// TwinCAT 3 PLC project Untitled1
// ProgramVersion: 3.1.4023.0
// libraries:
//   Tc2_Standard, * (Beckhoff Automation GmbH)
//   Tc2_System, * (Beckhoff Automation GmbH)
//   Tc3_Module, * (Beckhoff Automation GmbH)
// project tree:
//   DUTs/ ST_Banner_K30PTKQ_Control.TcDUT, ST_Banner_K30PTKQ_Status.TcDUT, ST_Keyence_LRXH100_Status.TcDUT, ST_Balluff_BMF00LA_Status.TcDUT
//   FBs/ FB_Banner_K30PTKQ.TcPOU, FB_Keyence_LRXH100.TcPOU, FB_Balluff_BMF00LA.TcPOU
//   / PlcTask.TcTTO
//   POUs/ MAIN.TcPOU

CONFIGURATION Untitled1
    RESOURCE PLC ON TwinCAT3
        TASK PlcTask(INTERVAL := T#10ms, PRIORITY := 20);
        PROGRAM MAIN WITH PlcTask : MAIN;
    END_RESOURCE
END_CONFIGURATION

// ---- DUTs/ST_Banner_K30PTKQ_Control.TcDUT
(*
	This structure contains all the inputs of the BANNER LED.
	The inputs and the outputs are linked to the device as well.
*)

TYPE ST_Banner_K30PTKQ_Control :
	STRUCT
	Color1					: UINT; (* 0 = Green, 1 = Red, 2 = Orange, 3 = Amber, 4 = Yellow,
									5 = Lime Green, 6 = Spring Green, 7 = Cyan, 8 = Sky Blue,
									9 = Blue, 10 = Violet, 11 = Magenta, 12 = Rose, 13 = White,
									14 = Custom1, 15 = Custom2 *)
	Color2					: UINT; (* 0 = Green, 1 = Red, 2 = Orange, 3 = Amber, 4 = Yellow,
									5 = Lime Green, 6 = Spring Green, 7 = Cyan, 8 = Sky Blue,
									9 = Blue, 10 = Violet, 11 = Magenta, 12 = Rose, 13 = White,
									14 = Custom1, 15 = Custom2 *)
	Color1Intensity			: UINT; (* 0 = High, 1 = Medium, 2 = Low, 3 = Off, 4 = Custom *)
	Color2Intensity			: UINT; (* 0 = High, 1 = Medium, 2 = Low, 3 = Off, 4 = Custom *)
	SequenceStartLocation	: UINT; (* 0 = LED1, 1 = LED2, 2 = LED3, 3 = LED4 *)
	DynamicSequenceValue	: UINT; (* 0-255 *)
	AnimationSpeed			: UINT; (* 0 = Slow, 1 = Medium, 2 = Fast, 3 = Custom *)
	Reserved				: UINT; (* Reserved *)
	AnimationType			: UINT; (* 0 = Off, 1 = Steady, 2 = Flash, 3 = Two Color Flash,
									   4 = 50/50, 5 = 50/50 Rotate, 6 = Chase, 7 = Intensity Sweep,
									   8 = Color Sweep, 9 = Sequence, 10 = Wave, 11 = Double Wave *)
	AnimationDirection		: UINT; (* 0 = CCW, 1 = CW *)
	AnimationPattern		: UINT; (* 0 = Flash, 1 = Strobe, 2 = Three Pulse, 3 = SOS, 4 = Random *)
	END_STRUCT
END_TYPE

// ---- DUTs/ST_Banner_K30PTKQ_Status.TcDUT
(*
	This structure contains all the outputs of the BANNER LED.
	The inputs and the outputs are linked to the device as well.
*)
TYPE ST_Banner_K30PTKQ_Status :
	STRUCT
	OutputState	: UINT; (* 0 = Normally Closed, 1 = Normally Open *)
	END_STRUCT
END_TYPE

// ---- DUTs/ST_Keyence_LRXH100_Status.TcDUT
(*
	This structure contains all the outputs of the BANNER LED.
	The inputs and the outputs are linked to the device as well.
*)
TYPE ST_Keyence_LRXH100_Status :
STRUCT
	CurrentValue		: INT; (* The distance from the target -9999 to 10001 *)
	ErrorOvercurrent	: BOOL; (* 0x7710 An overcurrent error has occurred. *)
	ErrorHeadError		: BOOL; (* 0x1803 A laser fault has occurred. *)
	ErrorEepromError	: BOOL; (* 0x5000 An EEPROM error has occurred in the sensor. *)
	Error17Error		: BOOL; (* 0x1807 Error 1 - 7 *)
	Output1				: BOOL; (* Output 1 *)
	Output2				: BOOL; (* Output 2 *)
	Warning				: BOOL; (* Warning *)
END_STRUCT
END_TYPE

// ---- DUTs/ST_Balluff_BMF00LA_Status.TcDUT
(*
	This structure contains all the outputs of the BANNER LED.
	The inputs and the outputs are linked to the device as well.
*)
TYPE ST_Balluff_BMF00LA_Status :
STRUCT
	Stability	: BOOL; (* Monitor if the sensor recognises a signal *)
	TeachIn		: BOOL; (* Monitor whether it is currently being taught *)
	BDC1		: BOOL; (* Setted point 1 *)
	BDC2		: BOOL; (* Setted point 2 *)
	BDC3		: BOOL; (* Setted point 3 *)
	BDC4		: BOOL; (* Setted point 4 *)
	BDC5		: BOOL; (* Setted point 5 *)
	BDC6		: BOOL; (* Setted point 6 *)
	BDC7		: BOOL; (* Setted point 7 *)
	BDC8		: BOOL; (* Setted point 8 *)
END_STRUCT
END_TYPE

// ---- POUs/MAIN.TcPOU
PROGRAM MAIN
VAR
{attribute 'TcLinkToOSO' := '.In.OutputState 			:= <0,1,0>TIID^Device 2 (EtherCAT)^Box 1 (EP6228-0022)^Banner_K30PTKQ^In^Output State;
							 .Out.Color1 	 			:= <0,5,0>TIID^Device 2 (EtherCAT)^Box 1 (EP6228-0022)^Banner_K30PTKQ^Out^Color 1;
							 .Out.Color2 	 			:= <0,5,0>TIID^Device 2 (EtherCAT)^Box 1 (EP6228-0022)^Banner_K30PTKQ^Out^Color 2;
							 .Out.Color1Intensity 	 	:= <0,3,0>TIID^Device 2 (EtherCAT)^Box 1 (EP6228-0022)^Banner_K30PTKQ^Out^Color 1 Intensity;
							 .Out.Color2Intensity 	 	:= <0,3,0>TIID^Device 2 (EtherCAT)^Box 1 (EP6228-0022)^Banner_K30PTKQ^Out^Color 2 Intensity;
							 .Out.SequenceStartLocation	:= <0,3,0>TIID^Device 2 (EtherCAT)^Box 1 (EP6228-0022)^Banner_K30PTKQ^Out^Sequence Start Location;
							 .Out.DynamicSequenceValue 	:= <0,8,0>TIID^Device 2 (EtherCAT)^Box 1 (EP6228-0022)^Banner_K30PTKQ^Out^Dynamic Sequence Value (0-255);
							 .Out.AnimationSpeed 	 	:= <0,2,0>TIID^Device 2 (EtherCAT)^Box 1 (EP6228-0022)^Banner_K30PTKQ^Out^Animation Speed;
							 .Out.Reserved 	 			:= <0,2,0>TIID^Device 2 (EtherCAT)^Box 1 (EP6228-0022)^Banner_K30PTKQ^Out^Reserved;
							 .Out.AnimationType 	 	:= <0,4,0>TIID^Device 2 (EtherCAT)^Box 1 (EP6228-0022)^Banner_K30PTKQ^Out^Animation Type;
							 .Out.AnimationDirection 	:= <0,1,0>TIID^Device 2 (EtherCAT)^Box 1 (EP6228-0022)^Banner_K30PTKQ^Out^Animation Direction;
							 .Out.AnimationPattern 	 	:= <0,3,0>TIID^Device 2 (EtherCAT)^Box 1 (EP6228-0022)^Banner_K30PTKQ^Out^Animation Pattern'}	
	LED		: FB_Banner_K30PTKQ; (*This is an instance of the FB_LED Funciton block*)
	{attribute 'TcLinkTo' := '.In.Stability 			:= TIID^Device 2 (EtherCAT)^Box 1 (EP6228-0022)^Balluff_BMF00LA^In^Stability;
							  .In.TeachIn 				:= TIID^Device 2 (EtherCAT)^Box 1 (EP6228-0022)^Balluff_BMF00LA^In^Teach-In;
							  .In.BDC1 					:= TIID^Device 2 (EtherCAT)^Box 1 (EP6228-0022)^Balluff_BMF00LA^In^BDC1;
							  .In.BDC2 					:= TIID^Device 2 (EtherCAT)^Box 1 (EP6228-0022)^Balluff_BMF00LA^In^BDC2;
							  .In.BDC3 					:= TIID^Device 2 (EtherCAT)^Box 1 (EP6228-0022)^Balluff_BMF00LA^In^BDC3;
							  .In.BDC4 					:= TIID^Device 2 (EtherCAT)^Box 1 (EP6228-0022)^Balluff_BMF00LA^In^BDC4;
							  .In.BDC5 					:= TIID^Device 2 (EtherCAT)^Box 1 (EP6228-0022)^Balluff_BMF00LA^In^BDC5;
							  .In.BDC6 					:= TIID^Device 2 (EtherCAT)^Box 1 (EP6228-0022)^Balluff_BMF00LA^In^BDC6;
							  .In.BDC7 					:= TIID^Device 2 (EtherCAT)^Box 1 (EP6228-0022)^Balluff_BMF00LA^In^BDC7;
							  .In.BDC8 					:= TIID^Device 2 (EtherCAT)^Box 1 (EP6228-0022)^Balluff_BMF00LA^In^BDC8'}
	Sensor	: FB_Balluff_BMF00LA; (*This is an instance of the FB_Sensor Funciton block*)
	
	{attribute 'TcLinkTo' := '.In.CurrentValue 			:= TIID^Device 2 (EtherCAT)^Box 1 (EP6228-0022)^Keyence_LRXH100^In^Current Value;
							  .In.ErrorOvercurrent 		:= TIID^Device 2 (EtherCAT)^Box 1 (EP6228-0022)^Keyence_LRXH100^In^Error : Overcurrent;
						      .In.ErrorHeadError	 	:= TIID^Device 2 (EtherCAT)^Box 1 (EP6228-0022)^Keyence_LRXH100^In^Error : Head Error;
							  .In.ErrorEepromError 	 	:= TIID^Device 2 (EtherCAT)^Box 1 (EP6228-0022)^Keyence_LRXH100^In^Error : EEPROM Error;
							  .In.Error17Error 			:= TIID^Device 2 (EtherCAT)^Box 1 (EP6228-0022)^Keyence_LRXH100^In^Error : Error 1 - 7;
							  .In.Output1 	 			:= TIID^Device 2 (EtherCAT)^Box 1 (EP6228-0022)^Keyence_LRXH100^In^Output 1;
							  .In.Output2	 	 		:= TIID^Device 2 (EtherCAT)^Box 1 (EP6228-0022)^Keyence_LRXH100^In^Output 2;
							  .In.Warning 	 			:= TIID^Device 2 (EtherCAT)^Box 1 (EP6228-0022)^Keyence_LRXH100^In^Warning'}
	KeyenceSensor			: FB_Keyence_LRXH100; (*This is an instance of the FB_Keyence Funciton block*)
END_VAR
VAR
	sVendorName				: STRING(64);
	sVendorText				: STRING(64);
	bTrig					: BOOL;
	fbAdsRead				: Tc2_System.ADSREAD;
	i						: INT;
	sData					: ARRAY[0..3] OF STRING(64);
	nIndexOffset			: ARRAY[0..3] OF UDINT := [16#00100000, 16#00110000, 16#00120000, 16#00130000];
	state					: INT := 0;
END_VAR

FB_CALL(); (* This action call all of the Function blocks *)
(* This function block makes the LED Interacting with the Keyence sensor *)
LED(
	nDistance:= KeyenceSensor.nDistance,
	nLowLimit:= 600,
	nHighLimit:= 1000);
			
(*IF bTrig THEN
	FOR i:=0 TO 3 BY 1 DO
		fbAdsRead(
			NETID	:= '10.62.25.99.3.2', 
			PORT	:= 16#1007, 
			IDXGRP	:= 16#F302,
			IDXOFFS	:= nIndexOffset[i], 
			LEN		:= SIZEOF(sData[i]), 
			DESTADDR:= ADR(sData[i]),
			READ	:= TRUE,
			TMOUT	:= T#3S);
	END_FOR
END_IF*)

(*IF bTrig THEN
	state 	:= 0;
	i 		:= 0;
	FOR i:=0 TO 3 BY 1 DO
		CASE state OF
			0:	// Init
				IF i=4 THEN
					bTrig := FALSE;
					RETURN;
				ELSE
					fbAdsRead(
						IDXOFFS	:= nIndexOffset[i], 
						LEN		:= SIZEOF(sData[i]), 
						DESTADDR:= ADR(sData[i]), 
						READ:= FALSE);
					
					MEMSET(ADR(sData[i]), 0, SIZEOF(sData[i]));
					state := state + 1;					
				END_IF

			1:	// Execute
					fbAdsRead(READ	:= TRUE);
					
					IF fbAdsRead.BUSY THEN
						state := state + 1;
					END_IF
				
			2:	// Done
				IF NOT fbAdsRead.BUSY THEN
					fbAdsRead(READ:= FALSE);
					state := 0;
				END_IF		
		END_CASE
	END_FOR
END_IF*)


//IF fbAdsRead.BUSY THEN
//	bTrig := FALSE;
//END_IF

ACTION FB_CALL:
KeyenceSensor();
Sensor();
LED();
END_ACTION

END_PROGRAM

// ---- FBs/FB_Banner_K30PTKQ.TcPOU
(*This Function block is for the BANNER LED*)
FUNCTION_BLOCK FB_Banner_K30PTKQ
VAR_INPUT
	nDistance	: INT;					(* The sensor actual distance from the targeted item *)
	nLowLimit	: INT := 200; 			(* The minimum distance of the valid intervall*)
	nHighLimit	: INT := 1200; 			(* The maximum distance of the valid intervall*)
END_VAR
VAR
	In		AT %I* 	: ST_Banner_K30PTKQ_Status;  (*THIS is an instance of the ST_BannerStatus STRUCTURE.*)
	Out 	AT %Q* 	: ST_Banner_K30PTKQ_Control;	(*THIS is an instance of the ST_BannerControl STRUCTURE.*)
	color1 			: UINT := 4;		(*0 = Green, 1 = Red, 2 = Orange, 3 = Amber, 4 = Yellow,
										5 = Lime Green, 6 = Spring Green, 7 = Cyan, 8 = Sky Blue,
										9 = Blue, 10 = Violet, 11 = Magenta, 12 = Rose, 13 = White,
										14 = Custom1, 15 = Custom2*)
	color2			: UINT := 1;		(*0 = Green, 1 = Red, 2 = Orange, 3 = Amber, 4 = Yellow,
										5 = Lime Green, 6 = Spring Green, 7 = Cyan, 8 = Sky Blue,
										9 = Blue, 10 = Violet, 11 = Magenta, 12 = Rose, 13 = White,
										14 = Custom1, 15 = Custom2*)
END_VAR

(* If the targeted distance is optimal the Banner is Green else it is red.
If the distance is too big or too small the banner is off *)
IF nDistance <> 10000 THEN
	IF nDistance <= nLowLimit OR nDistance >= nHighLimit THEN
		Out.Color1 := 1;
		Out.Color2 := 1;
		Out.Color2Intensity := 2;
		Out.AnimationType	:= 10;
		Out.AnimationSpeed := 1;
	ELSE
		Out.Color1 := 0;
		Out.Color2 := 0;
		Out.Color2Intensity := 2;
		Out.AnimationType	:= 10;
		Out.AnimationSpeed := 1;	
	END_IF
ELSE
	Out.Color1 := 1;
	Out.Color2 := 1;
	Out.Color2Intensity := 2;
	Out.AnimationType	:= 0;
	Out.AnimationSpeed := 1;
END_IF

END_FUNCTION_BLOCK

// ---- FBs/FB_Balluff_BMF00LA.TcPOU
(* This Function block is for the BALLUF sensor *)
FUNCTION_BLOCK FB_Balluff_BMF00LA
VAR
	In		AT %I* 	: ST_Balluff_BMF00LA_Status;
END_VAR

END_FUNCTION_BLOCK

// ---- FBs/FB_Keyence_LRXH100.TcPOU
(* This Function block is for the Keyence sensor *)
FUNCTION_BLOCK FB_Keyence_LRXH100
VAR_OUTPUT
	nDistance	: INT;
END_VAR
VAR
	In	AT %I*	: ST_Keyence_LRXH100_Status;
END_VAR

(* Setting the output value to the current distance *)
nDistance := In.CurrentValue;

END_FUNCTION_BLOCK
